FUNCTION_BLOCK Velocity_PI_ACC (* Composite Function Block Type *)
  (* Standard: 61499-2 *)
  (* Version 0.0, 2018-07-28, 4DIAC-IDE, 4DIAC-Consortium *)
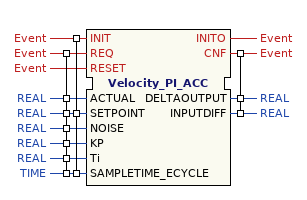
  EVENT_INPUT
    INIT WITH SAMPLETIME_ECYCLE, SETPOINT; (* Initialization Request *)
    REQ WITH ACTUAL, SETPOINT, NOISE, KP, SAMPLETIME_ECYCLE, Ti; (* Normal Execution Request. disambung Event Cycle juga ya *)
    RESET;
  END_EVENT
  EVENT_OUTPUT
    INITO; (* Initialization Confirm *)
    CNF WITH DELTAOUTPUT, INPUTDIFF; (* Execution Confirmation *)
  END_EVENT
  VAR_INPUT
    ACTUAL : REAL;
    SETPOINT : REAL;
    NOISE : REAL;
    KP : REAL;
    Ti : REAL;
    SAMPLETIME_ECYCLE : TIME;
  END_VAR
  VAR_OUTPUT
    DELTAOUTPUT : REAL;
    INPUTDIFF : REAL;
  END_VAR
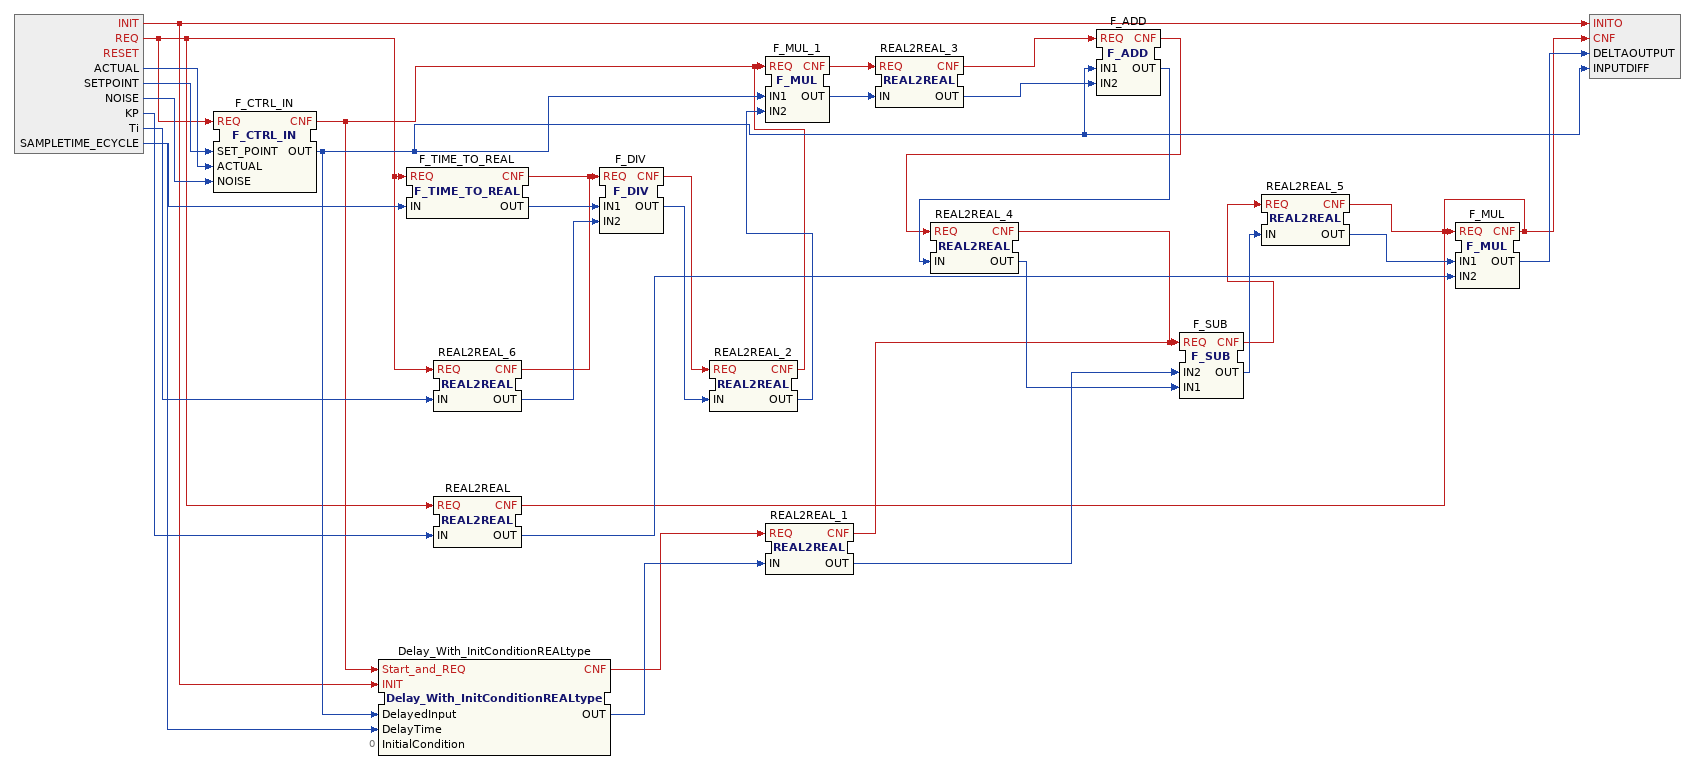
  FBS
    F_CTRL_IN : F_CTRL_IN;
    REAL2REAL : REAL2REAL;
    F_SUB : F_SUB;
    Delay_With_InitConditionREALtype : Delay_With_InitConditionREALtype(InitialCondition := 0);
    F_MUL : F_MUL;
    REAL2REAL_1 : REAL2REAL;
    F_ADD : F_ADD;
    F_MUL_1 : F_MUL;
    F_TIME_TO_REAL : F_TIME_TO_REAL;
    F_DIV : F_DIV;
    REAL2REAL_2 : REAL2REAL;
    REAL2REAL_3 : REAL2REAL;
    REAL2REAL_4 : REAL2REAL;
    REAL2REAL_5 : REAL2REAL;
    REAL2REAL_6 : REAL2REAL;
  END_FBS
  EVENT_CONNECTIONS
    REQ TO F_CTRL_IN.REQ;
    REAL2REAL_1.CNF TO F_SUB.REQ;
    F_CTRL_IN.CNF TO Delay_With_InitConditionREALtype.Start_and_REQ;
    INIT TO Delay_With_InitConditionREALtype.INIT;
    REQ TO REAL2REAL.REQ;
    Delay_With_InitConditionREALtype.CNF TO REAL2REAL_1.REQ;
    REAL2REAL_4.CNF TO F_SUB.REQ;
    F_ADD.CNF TO REAL2REAL_4.REQ;
    REAL2REAL_3.CNF TO F_ADD.REQ;
    F_MUL_1.CNF TO REAL2REAL_3.REQ;
    F_TIME_TO_REAL.CNF TO F_DIV.REQ;
    REQ TO F_TIME_TO_REAL.REQ;
    F_CTRL_IN.CNF TO F_MUL_1.REQ;
    F_DIV.CNF TO REAL2REAL_2.REQ;
    REAL2REAL_2.CNF TO F_MUL_1.REQ;
    F_SUB.CNF TO REAL2REAL_5.REQ;
    REAL2REAL_5.CNF TO F_MUL.REQ;
    F_MUL.CNF TO CNF;
    REAL2REAL.CNF TO F_MUL.REQ;
    F_MUL.CNF TO F_MUL.REQ;
    INIT TO INITO;
    REAL2REAL_6.CNF TO F_DIV.REQ;
    REQ TO REAL2REAL_6.REQ;
  END_CONNECTIONS
  DATA_CONNECTIONS
    KP TO REAL2REAL.IN;
    F_CTRL_IN.OUT TO INPUTDIFF;
    F_CTRL_IN.OUT TO Delay_With_InitConditionREALtype.DelayedInput;
    SETPOINT TO F_CTRL_IN.SET_POINT;
    ACTUAL TO F_CTRL_IN.ACTUAL;
    NOISE TO F_CTRL_IN.NOISE;
    REAL2REAL_1.OUT TO F_SUB.IN2;
    F_CTRL_IN.OUT TO F_ADD.IN1;
    F_CTRL_IN.OUT TO F_MUL_1.IN1;
    SAMPLETIME_ECYCLE TO Delay_With_InitConditionREALtype.DelayTime;
    F_TIME_TO_REAL.OUT TO F_DIV.IN1;
    SAMPLETIME_ECYCLE TO F_TIME_TO_REAL.IN;
    F_DIV.OUT TO REAL2REAL_2.IN;
    REAL2REAL_2.OUT TO F_MUL_1.IN2;
    F_MUL_1.OUT TO REAL2REAL_3.IN;
    REAL2REAL_3.OUT TO F_ADD.IN2;
    REAL2REAL_4.OUT TO F_SUB.IN1;
    F_ADD.OUT TO REAL2REAL_4.IN;
    Delay_With_InitConditionREALtype.OUT TO REAL2REAL_1.IN;
    F_SUB.OUT TO REAL2REAL_5.IN;
    REAL2REAL_5.OUT TO F_MUL.IN1;
    REAL2REAL.OUT TO F_MUL.IN2;
    F_MUL.OUT TO DELTAOUTPUT;
    REAL2REAL_6.OUT TO F_DIV.IN2;
    Ti TO REAL2REAL_6.IN;
  END_CONNECTIONS
END_FUNCTION_BLOCK
